// Minimal I_Telescope that only records what the MQTT handler asks it to do.
FUNCTION_BLOCK FB_TelescopeStub IMPLEMENTS BROTLib.I_Telescope
VAR_OUTPUT
	nTrack			: INT;		// number of Track() calls
	fTrackRa		: LREAL;	// arguments of the last Track()
	fTrackDec		: LREAL;
	nSlew			: INT;		// number of Slew() calls
	fSlewAz			: LREAL;	// arguments of the last Slew()
	fSlewAlt		: LREAL;
	nOther			: INT;		// Home / Init / Park / Reset / Stop calls
END_VAR
VAR
	bCoverAutoOpen	: BOOL;
END_VAR

METHOD ClearCounters : BOOL
VAR_INPUT
END_VAR
nTrack := 0; fTrackRa := 0.0; fTrackDec := 0.0;
nSlew := 0; fSlewAz := 0.0; fSlewAlt := 0.0;
nOther := 0;
ClearCounters := TRUE;
END_METHOD

METHOD Home : BOOL
VAR_INPUT
END_VAR
nOther := nOther + 1;
Home := TRUE;
END_METHOD

METHOD Init : BOOL
VAR_INPUT
END_VAR
nOther := nOther + 1;
Init := TRUE;
END_METHOD

METHOD Park : BOOL
VAR_INPUT
END_VAR
nOther := nOther + 1;
Park := TRUE;
END_METHOD

METHOD Reset : BOOL
VAR_INPUT
END_VAR
nOther := nOther + 1;
Reset := TRUE;
END_METHOD

METHOD Stop : BOOL
VAR_INPUT
END_VAR
nOther := nOther + 1;
Stop := TRUE;
END_METHOD

METHOD Slew : BOOL
VAR_INPUT
	fAzimuth	: LREAL;
	fAltitude	: LREAL;
END_VAR
nSlew := nSlew + 1;
fSlewAz := fAzimuth;
fSlewAlt := fAltitude;
Slew := TRUE;
END_METHOD

METHOD Track : BOOL
VAR_INPUT
	fRightAscension	: LREAL;
	fDeclination	: LREAL;
END_VAR
nTrack := nTrack + 1;
fTrackRa := fRightAscension;
fTrackDec := fDeclination;
Track := TRUE;
END_METHOD

PROPERTY Altitude : LREAL
GET
Altitude := fSlewAlt;
END_GET
END_PROPERTY

PROPERTY Azimuth : LREAL
GET
Azimuth := fSlewAz;
END_GET
END_PROPERTY

PROPERTY Declination : LREAL
GET
Declination := fTrackDec;
END_GET
END_PROPERTY

PROPERTY RightAscension : LREAL
GET
RightAscension := fTrackRa;
END_GET
END_PROPERTY

PROPERTY CoverAutoOpen : BOOL
GET
CoverAutoOpen := bCoverAutoOpen;
END_GET
SET
bCoverAutoOpen := CoverAutoOpen;
END_SET
END_PROPERTY

END_FUNCTION_BLOCK

(* stored: Version 1.1.0.1, ProductVersion 3.1.4024.15
   POU FB_TelescopeStub: Id {94896858-e375-45fa-8185-d6e1eb0e6752}, SpecialFunc None
   Method ClearCounters: Id {dbed822d-5ef7-4e4c-879b-8489f044a9c3}
   Method Home: Id {a576499b-e0e7-4b0a-b36c-d18d1cf2465c}
   Method Init: Id {36312c01-6a95-462f-b0b7-06307001967a}
   Method Park: Id {094c25e1-a33b-4906-81cd-86ad398b3b46}
   Method Reset: Id {b4aefd18-a438-4adb-ac4f-e4396a08a9a0}
   Method Stop: Id {3e1444b8-464e-459f-a4a7-4c693d816795}
   Method Slew: Id {52302751-cb70-4524-9cf9-3f472cf20eb5}
   Method Track: Id {5aa3ca1c-0cf1-4a57-8ea3-44ca09468218}
   Property Altitude: Id {06212c45-5841-4ad4-812d-331b3ee572b0}
   Get Get: Id {691eb4c8-da5b-4c1c-a788-b422685f0037}
   Property Azimuth: Id {8c8f752e-c3e6-477f-b2c1-f6531d3cbf2b}
   Get Get: Id {57a86085-e7dc-4b5e-bf9c-b698ba20ecfd}
   Property Declination: Id {24caef07-e8df-4d8e-99f0-6fba5bb9b6a0}
   Get Get: Id {01f1bec2-91f3-4f4d-8aa3-e8771b7e907d}
   Property RightAscension: Id {97b9bc6b-cce8-467a-bc5c-0226b8b22337}
   Get Get: Id {532f6d71-1748-4ca8-9122-a33953968cc6}
   Property CoverAutoOpen: Id {3282ebb7-57b9-4bd4-9b20-2d73243eaef5}
   Get Get: Id {5c19cb3c-52e4-494d-b407-1ffe70da1e35}
   Set Set: Id {6aab54b9-dc2b-4451-bee2-007d1a8bf795} *)
